(* PLC project KinIn_v3.project, CODESYS CODESYS V3.5 SP19 *)
(* stored: creationDateTime 2025-01-20T16:18:42.0738422, modificationDateTime 2025-01-20T16:17:39.6822999 *)

FUNCTION_BLOCK Inv
  VAR_INPUT
    matSquare : ARRAY[1..GVL.nInvSize, 1..GVL.nInvSize] OF REAL;
  END_VAR
  VAR_OUTPUT
    InverseMatrix : ARRAY[1..GVL.nInvSize, 1..GVL.nInvSize] OF REAL;
  END_VAR
  VAR
    LuDecomposition : LuDecomposition;
    Eye : Eye;
    LuInverse : LuInverse;
    L : ARRAY[1..GVL.nInvSize, 1..GVL.nInvSize] OF REAL;  (* LU factor same size input matrix *)
    U : ARRAY[1..GVL.nInvSize, 1..GVL.nInvSize] OF REAL;
    d : ARRAY[1..GVL.nInvSize, 1..GVL.nInvSize] OF REAL;
    eyeN : ARRAY[1..GVL.nInvSize, 1..GVL.nInvSize] OF REAL;
  END_VAR

            LuDecomposition(A:=matSquare , 
		L:= L, U:= U);
		
Eye(eye:= eyeN);

LuInverse(
	L:= L, 
	u:= U, 
	a:= InverseMatrix, 
	d:= d, 
	eyeN:= eyeN);
          
END_FUNCTION_BLOCK
